// Mitsubishi GX Works2 project: X27   PLC: FX3G

// task Task_01 (event TRUE, interval 0, priority 31): POU_01

PROGRAM POU_01
VAR
  wstep : INT;
  pwd : INT;
  inPwd : INT;
  rt1 : R_TRIG;
  rt2 : R_TRIG;
  ton1 : TON;
END_VAR
M99 := FALSE AND
M4 AND M5 AND M6 AND
Y1;

D0 := pwd;
D1 := inPwd;

IF M8002 THEN
    wstep := 0;
    pwd := 0;
    inPwd := 0;
END_IF;

rt1(_clk := M4);
rt2(_clk := M5);

CASE wstep OF
    0:
        IF rt1.q THEN
            IF (pwd + 10) >= 100 THEN
                pwd := pwd - 90;
            ELSE
                pwd := pwd + 10;
            END_IF;
        END_IF;
        IF rt2.q THEN
            IF (pwd MOD 10 + 1) >= 10 THEN
                pwd := pwd - 9;
            ELSE
                pwd := pwd + 1;
            END_IF;
        END_IF;

        IF M6 AND (pwd <> 0) THEN
            wstep := 1;
        END_IF;
    1:
    	Y1 := TRUE;
        IF rt1.q THEN
            IF (inPwd + 10) >= 100 THEN
                inPwd := inPwd - 90;
            ELSE
                inPwd := inPwd + 10;
            END_IF;
        END_IF;
        IF rt2.q THEN
            IF (inPwd MOD 10 + 1) >= 10 THEN
                inPwd := inPwd - 9;
            ELSE
                inPwd := inPwd + 1;
            END_IF;
        END_IF;

        IF M6 AND (inPwd <> 0) THEN
            wstep := 2;
        END_IF;
    2:
        Y1 := FALSE;
        IF pwd = inPwd THEN
            pwd := 0;
            inPwd := 0;
            wstep := 0;
        ELSE
            ton1(in := NOT ton1.q, pt := t#1.0s);
            inPwd := 0;

            IF ton1.q THEN
                wstep := 1;
            END_IF;
        END_IF;
END_CASE;
END_PROGRAM
